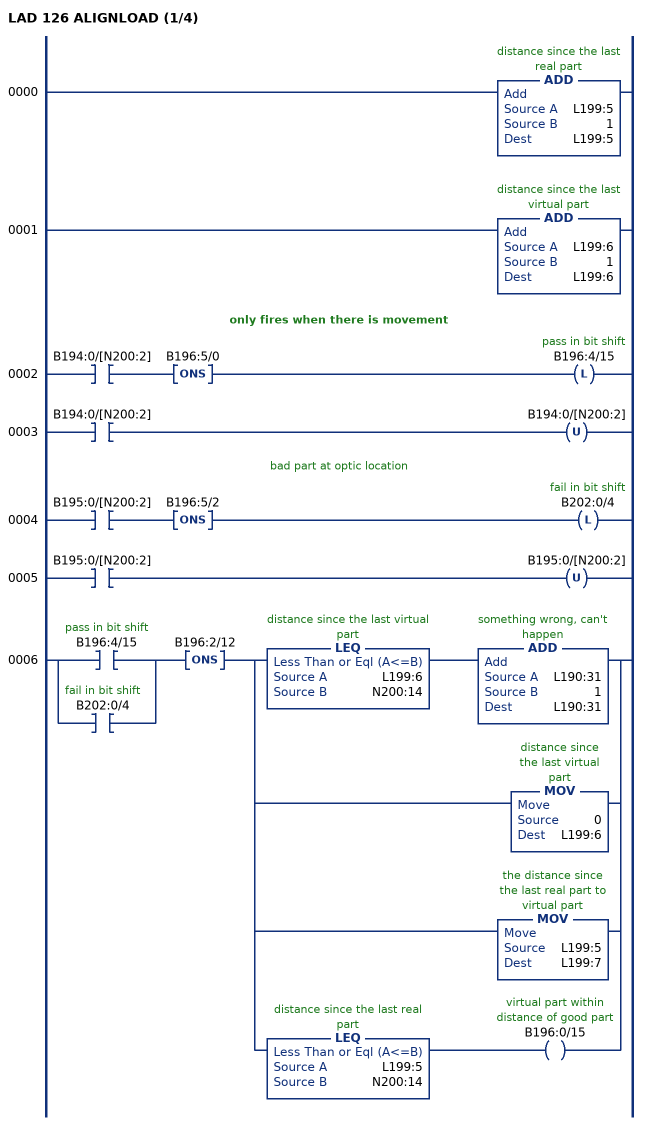
% Rung: 0 %
SOR ADD L199:5 1 L199:5 EOR
%   L199:5  "distance since the last real part" %
% Rung: 1 %
SOR ADD L199:6 1 L199:6 EOR
%   L199:6  "distance since the last virtual part" %
% Rung: 2 %
% TITLE: only fires when there is movement %
SOR XIC B194:0/[N200:2] ONS B196:5/0 OTL B196:4/15 EOR
%   N200:2  OPTIC_LOC  "top optic location" %
%   B196:4/15  "pass in bit shift" %
% Rung: 3 %
SOR XIC B194:0/[N200:2] OTU B194:0/[N200:2] EOR
%   N200:2  OPTIC_LOC  "top optic location" %
% Rung: 4 %
% bad part at optic location %
SOR XIC B195:0/[N200:2] ONS B196:5/2 OTL B202:0/4 EOR
%   N200:2  OPTIC_LOC  "top optic location" %
%   B202:0/4  "fail in bit shift" %
% Rung: 5 %
SOR XIC B195:0/[N200:2] OTU B195:0/[N200:2] EOR
%   N200:2  OPTIC_LOC  "top optic location" %
% Rung: 6 %
SOR BST XIC B196:4/15 NXB XIC B202:0/4 BND ONS B196:2/12 BST LEQ L199:6 N200:14 ADD L190:31 1 L190:31 NXB MOV 0 L199:6 NXB MOV L199:5 L199:7 NXB LEQ L199:5 N200:14 OTE B196:0/15 BND EOR
%   B196:4/15  "pass in bit shift" %
%   B202:0/4  "fail in bit shift" %
%   L199:6  "distance since the last virtual part" %
%   N200:14  "1/2 transistion zone" %
%   L190:31  "something wrong, can't happen" %
%   L199:5  "distance since the last real part" %
%   L199:7  "the distance since the last real part to virtual part" %
%   B196:0/15  "virtual part within distance of good part" %

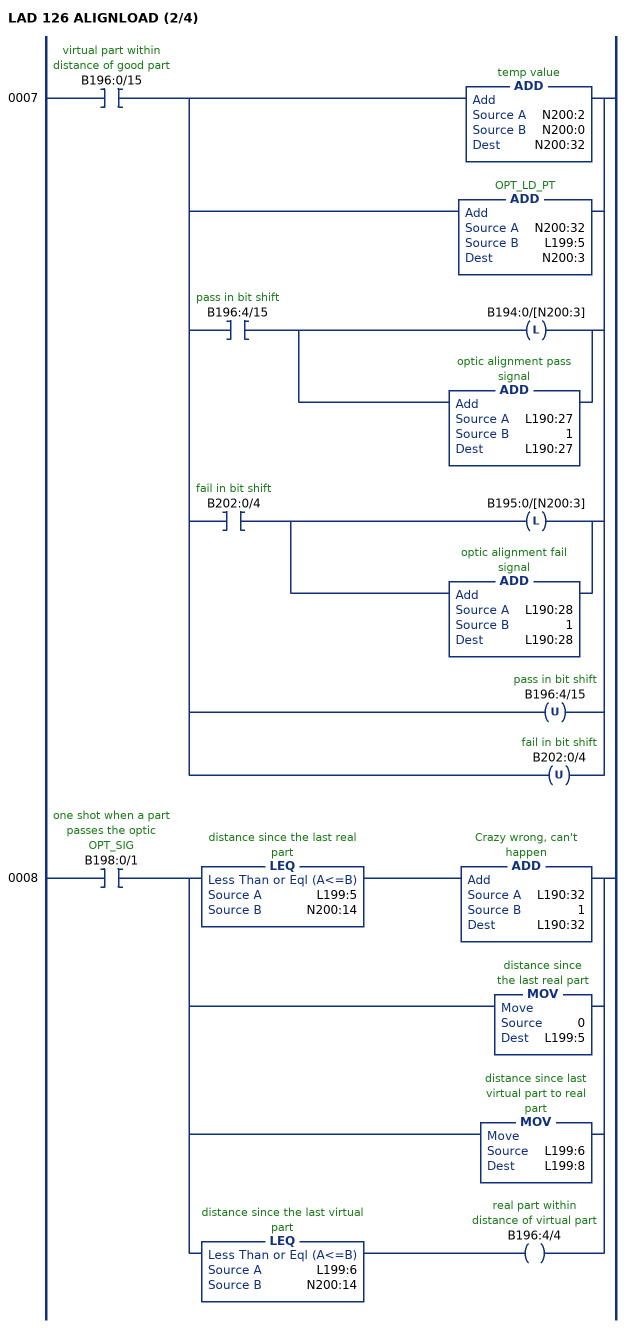
% Rung: 7 %
SOR XIC B196:0/15 BST ADD N200:2 N200:0 N200:32 NXB ADD N200:32 L199:5 N200:3 NXB XIC B196:4/15 BST OTL B194:0/[N200:3] NXB ADD L190:27 1 L190:27 BND NXB XIC B202:0/4 BST OTL B195:0/[N200:3] NXB ADD L190:28 1 L190:28 BND NXB OTU B196:4/15 NXB OTU B202:0/4 BND EOR
%   B196:0/15  "virtual part within distance of good part" %
%   N200:2  OPTIC_LOC  "top optic location" %
%   N200:0  PART_OFFSET  "1/2 part width" %
%   N200:32  "temp value" %
%   L199:5  "distance since the last real part" %
%   N200:3  OPT_LD_PT %
%   B196:4/15  "pass in bit shift" %
%   L190:27  "optic alignment pass signal" %
%   B202:0/4  "fail in bit shift" %
%   L190:28  "optic alignment fail signal" %
% Rung: 8 %
SOR XIC B198:0/1 BST LEQ L199:5 N200:14 ADD L190:32 1 L190:32 NXB MOV 0 L199:5 NXB MOV L199:6 L199:8 NXB LEQ L199:6 N200:14 OTE B196:4/4 BND EOR
%   B198:0/1  OPT_SIG  "one shot when a part passes the optic" %
%   L199:5  "distance since the last real part" %
%   N200:14  "1/2 transistion zone" %
%   L190:32  "Crazy wrong, can't happen" %
%   L199:6  "distance since the last virtual part" %
%   L199:8  "distance since last virtual part to real part" %
%   B196:4/4  "real part within distance of virtual part" %

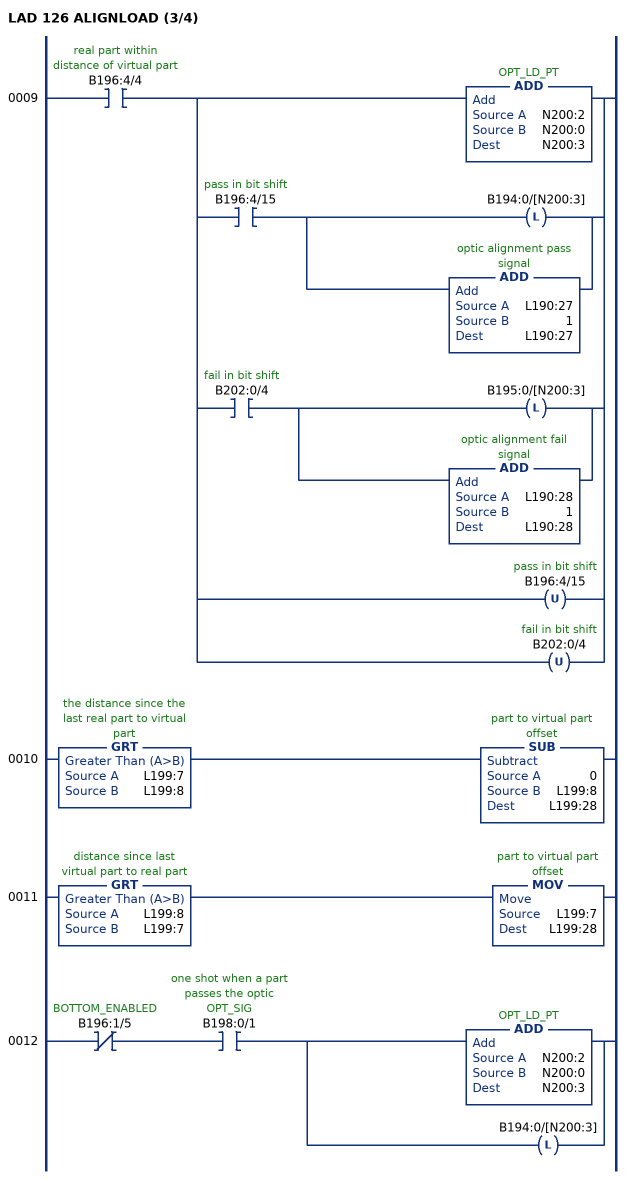
% Rung: 9 %
SOR XIC B196:4/4 BST ADD N200:2 N200:0 N200:3 NXB XIC B196:4/15 BST OTL B194:0/[N200:3] NXB ADD L190:27 1 L190:27 BND NXB XIC B202:0/4 BST OTL B195:0/[N200:3] NXB ADD L190:28 1 L190:28 BND NXB OTU B196:4/15 NXB OTU B202:0/4 BND EOR
%   B196:4/4  "real part within distance of virtual part" %
%   N200:2  OPTIC_LOC  "top optic location" %
%   N200:0  PART_OFFSET  "1/2 part width" %
%   N200:3  OPT_LD_PT %
%   B196:4/15  "pass in bit shift" %
%   L190:27  "optic alignment pass signal" %
%   B202:0/4  "fail in bit shift" %
%   L190:28  "optic alignment fail signal" %
% Rung: 10 %
SOR GRT L199:7 L199:8 SUB 0 L199:8 L199:28 EOR
%   L199:7  "the distance since the last real part to virtual part" %
%   L199:8  "distance since last virtual part to real part" %
%   L199:28  "part to virtual part offset" %
% Rung: 11 %
SOR GRT L199:8 L199:7 MOV L199:7 L199:28 EOR
%   L199:8  "distance since last virtual part to real part" %
%   L199:7  "the distance since the last real part to virtual part" %
%   L199:28  "part to virtual part offset" %
% Rung: 12 %
SOR XIO B196:1/5 XIC B198:0/1 BST ADD N200:2 N200:0 N200:3 NXB OTL B194:0/[N200:3] BND EOR
%   B196:1/5  BOTTOM_ENABLED %
%   B198:0/1  OPT_SIG  "one shot when a part passes the optic" %
%   N200:2  OPTIC_LOC  "top optic location" %
%   N200:0  PART_OFFSET  "1/2 part width" %
%   N200:3  OPT_LD_PT %

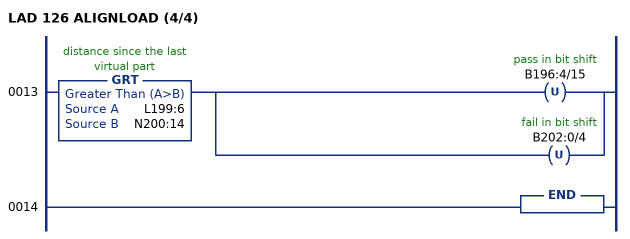
% Rung: 13 %
SOR GRT L199:6 N200:14 BST OTU B196:4/15 NXB OTU B202:0/4 BND EOR
%   L199:6  "distance since the last virtual part" %
%   N200:14  "1/2 transistion zone" %
%   B196:4/15  "pass in bit shift" %
%   B202:0/4  "fail in bit shift" %
% Rung: 14 %
SOR END EOR

LADDER 127 "NOTUSED"
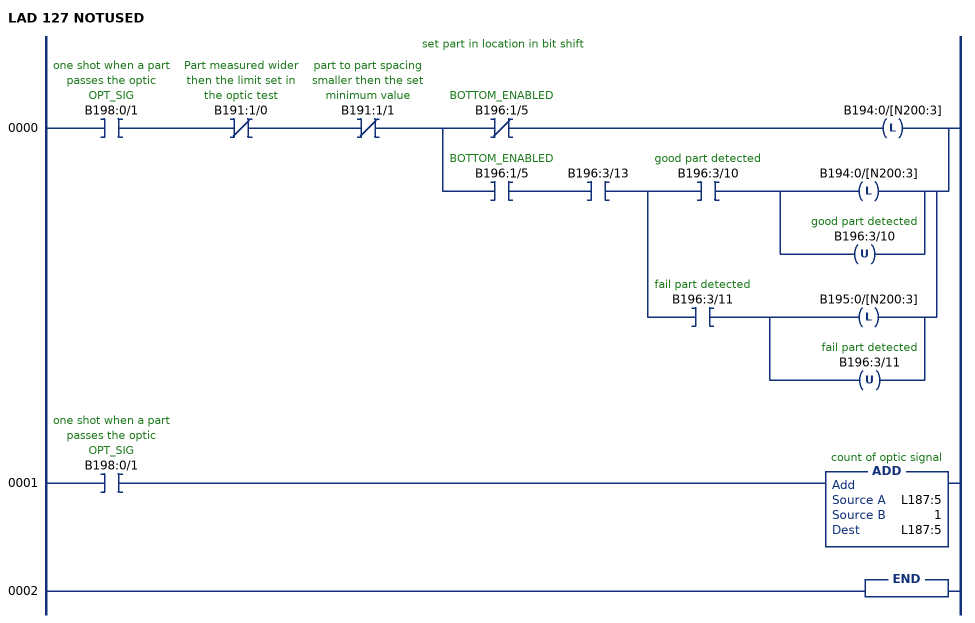
% Rung: 0 %
% set part in location in bit shift %
SOR XIC B198:0/1 XIO B191:1/0 XIO B191:1/1 BST XIO B196:1/5 OTL B194:0/[N200:3] NXB XIC B196:1/5 XIC B196:3/13 BST XIC B196:3/10 BST OTL B194:0/[N200:3] NXB OTU B196:3/10 BND NXB XIC B196:3/11 BST OTL B195:0/[N200:3] NXB OTU B196:3/11 BND BND BND EOR
%   B198:0/1  OPT_SIG  "one shot when a part passes the optic" %
%   B191:1/0  "Part measured wider then the limit set in the optic test" %
%   B191:1/1  "part to part spacing smaller then the set minimum value" %
%   B196:1/5  BOTTOM_ENABLED %
%   N200:3  OPT_LD_PT %
%   B196:3/10  "good part detected" %
%   B196:3/11  "fail part detected" %
% Rung: 1 %
SOR XIC B198:0/1 ADD L187:5 1 L187:5 EOR
%   B198:0/1  OPT_SIG  "one shot when a part passes the optic" %
%   L187:5  "count of optic signal" %
% Rung: 2 %
SOR END EOR

LADDER 128 "NOTUSED3"
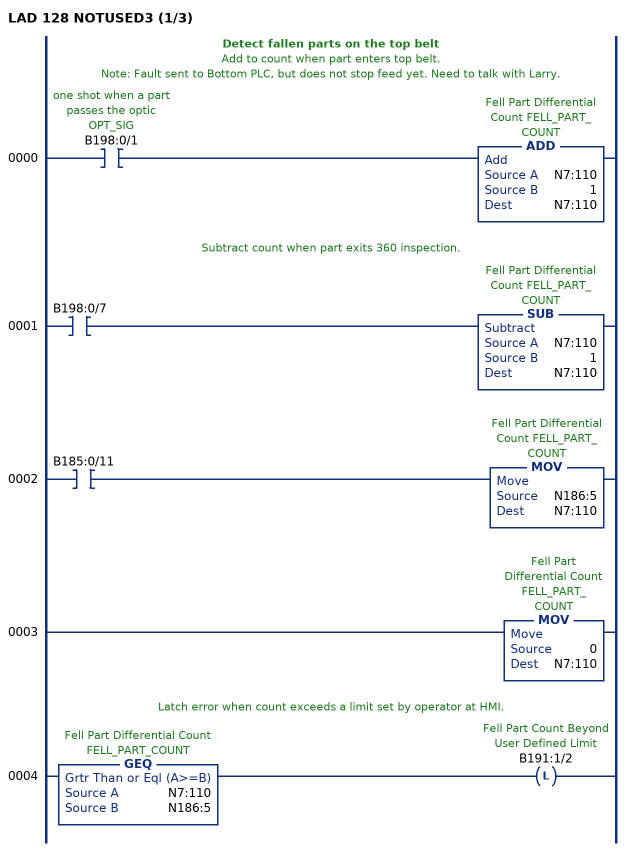
% Rung: 0 %
% TITLE: Detect fallen parts on the top belt %
% Add to count when part enters top belt.
% Note: Fault sent to Bottom PLC, but does not stop feed yet. Need to talk with Larry. %
SOR XIC B198:0/1 ADD N7:110 1 N7:110 EOR
%   B198:0/1  OPT_SIG  "one shot when a part passes the optic" %
%   N7:110  FELL_PART_COUNT  "Fell Part Differential Count" %
% Rung: 1 %
% Subtract count when part exits 360 inspection. %
SOR XIC B198:0/7 SUB N7:110 1 N7:110 EOR
%   N7:110  FELL_PART_COUNT  "Fell Part Differential Count" %
% Rung: 2 %
SOR XIC B185:0/11 MOV N186:5 N7:110 EOR
%   N186:5  FELL_PART_LIMIT  "Fell Part Differential Limit From HMI" %
%   N7:110  FELL_PART_COUNT  "Fell Part Differential Count" %
% Rung: 3 %
SOR MOV 0 N7:110 EOR
%   N7:110  FELL_PART_COUNT  "Fell Part Differential Count" %
% Rung: 4 %
% Latch error when count exceeds a limit set by operator at HMI. %
SOR GEQ N7:110 N186:5 OTL B191:1/2 EOR
%   N7:110  FELL_PART_COUNT  "Fell Part Differential Count" %
%   N186:5  FELL_PART_LIMIT  "Fell Part Differential Limit From HMI" %
%   B191:1/2  "Fell Part Count Beyond User Defined Limit" %

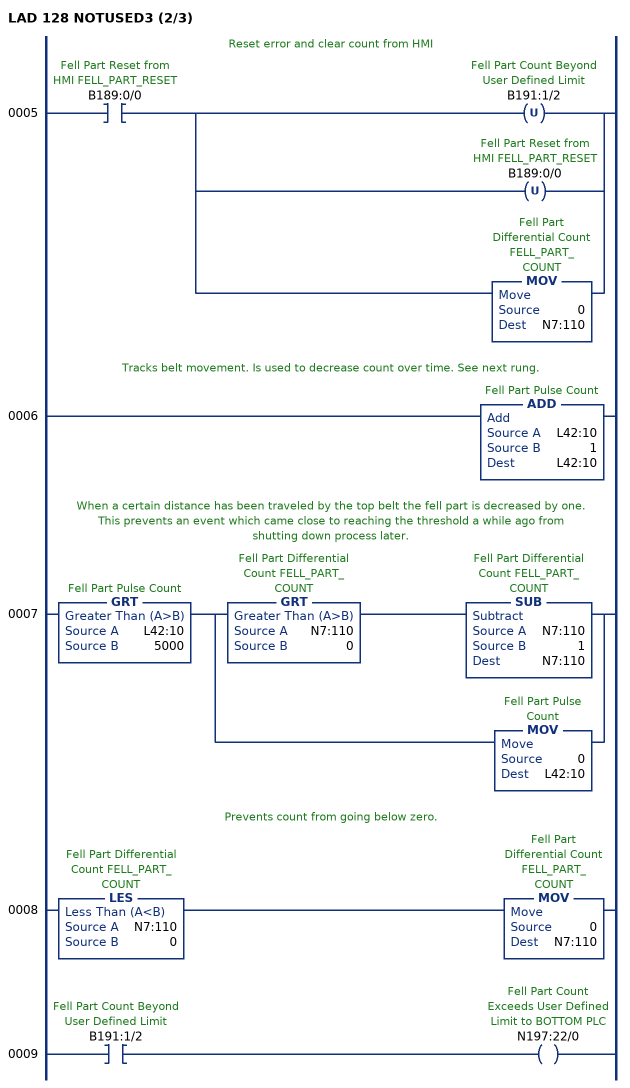
% Rung: 5 %
% Reset error and clear count from HMI %
SOR XIC B189:0/0 BST OTU B191:1/2 NXB OTU B189:0/0 NXB MOV 0 N7:110 BND EOR
%   B189:0/0  FELL_PART_RESET  "Fell Part Reset from HMI" %
%   B191:1/2  "Fell Part Count Beyond User Defined Limit" %
%   N7:110  FELL_PART_COUNT  "Fell Part Differential Count" %
% Rung: 6 %
% Tracks belt movement. Is used to decrease count over time. See next rung. %
SOR ADD L42:10 1 L42:10 EOR
%   L42:10  "Fell Part Pulse Count" %
% Rung: 7 %
% When a certain distance has been traveled by the top belt the fell part is decreased by one. This prevents an event which came close to reaching the threshold a while ago from shutting down process later. %
SOR GRT L42:10 5000 BST GRT N7:110 0 SUB N7:110 1 N7:110 NXB MOV 0 L42:10 BND EOR
%   L42:10  "Fell Part Pulse Count" %
%   N7:110  FELL_PART_COUNT  "Fell Part Differential Count" %
% Rung: 8 %
% Prevents count from going below zero. %
SOR LES N7:110 0 MOV 0 N7:110 EOR
%   N7:110  FELL_PART_COUNT  "Fell Part Differential Count" %
% Rung: 9 %
SOR XIC B191:1/2 OTE N197:22/0 EOR
%   B191:1/2  "Fell Part Count Beyond User Defined Limit" %
%   N197:22/0  "Fell Part Count Exceeds User Defined Limit to BOTTOM PLC" %

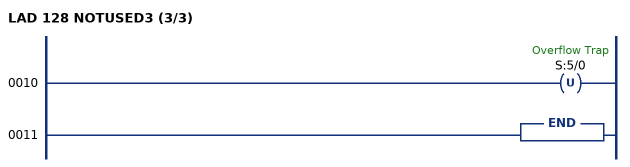
% Rung: 10 %
SOR OTU S:5/0 EOR
%   S:5/0  "Overflow Trap" %
% Rung: 11 %
SOR END EOR

LADDER 130 "INS 5 TRIG"
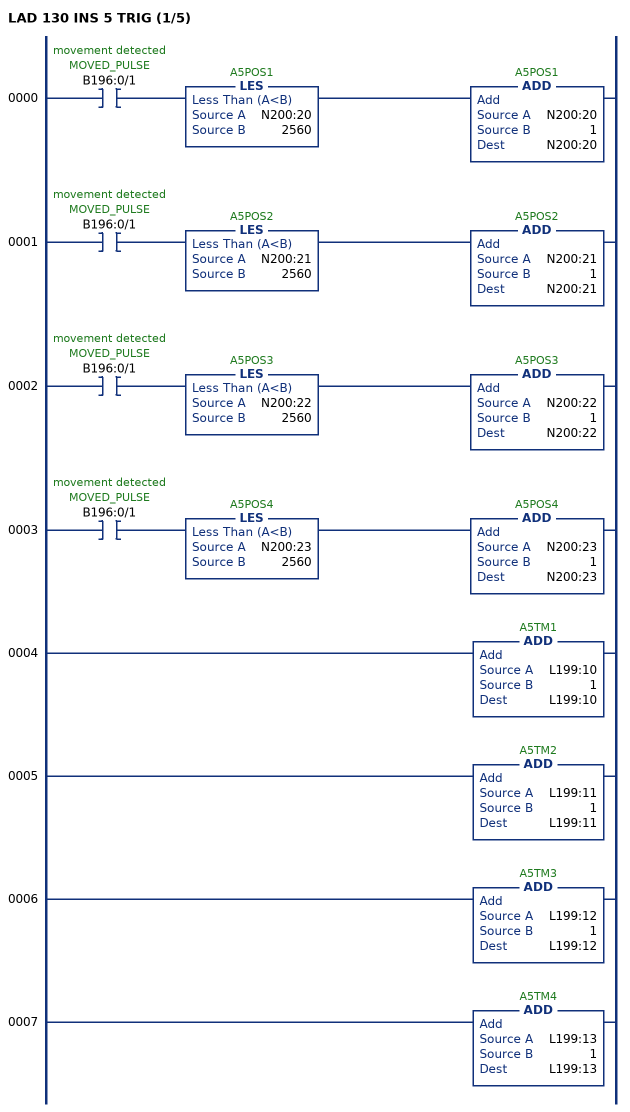
% Rung: 0 %
SOR XIC B196:0/1 LES N200:20 2560 ADD N200:20 1 N200:20 EOR
%   B196:0/1  MOVED_PULSE  "movement detected" %
%   N200:20  A5POS1 %
% Rung: 1 %
SOR XIC B196:0/1 LES N200:21 2560 ADD N200:21 1 N200:21 EOR
%   B196:0/1  MOVED_PULSE  "movement detected" %
%   N200:21  A5POS2 %
% Rung: 2 %
SOR XIC B196:0/1 LES N200:22 2560 ADD N200:22 1 N200:22 EOR
%   B196:0/1  MOVED_PULSE  "movement detected" %
%   N200:22  A5POS3 %
% Rung: 3 %
SOR XIC B196:0/1 LES N200:23 2560 ADD N200:23 1 N200:23 EOR
%   B196:0/1  MOVED_PULSE  "movement detected" %
%   N200:23  A5POS4 %
% Rung: 4 %
SOR ADD L199:10 1 L199:10 EOR
%   L199:10  A5TM1 %
% Rung: 5 %
SOR ADD L199:11 1 L199:11 EOR
%   L199:11  A5TM2 %
% Rung: 6 %
SOR ADD L199:12 1 L199:12 EOR
%   L199:12  A5TM3 %
% Rung: 7 %
SOR ADD L199:13 1 L199:13 EOR
%   L199:13  A5TM4 %

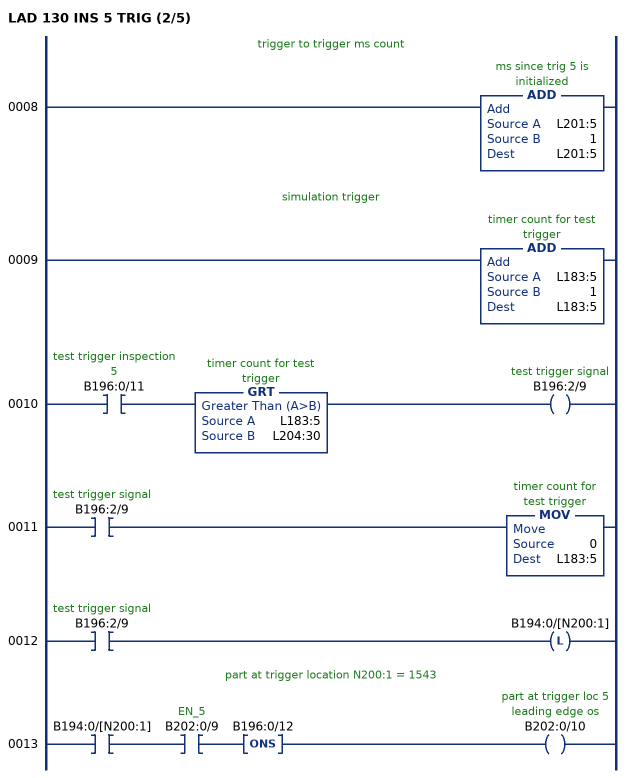
% Rung: 8 %
% trigger to trigger ms count %
SOR ADD L201:5 1 L201:5 EOR
%   L201:5  "ms since trig 5 is initialized" %
% Rung: 9 %
% simulation trigger %
SOR ADD L183:5 1 L183:5 EOR
%   L183:5  "timer count for test trigger" %
% Rung: 10 %
SOR XIC B196:0/11 GRT L183:5 L204:30 OTE B196:2/9 EOR
%   B196:0/11  "test trigger inspection 5" %
%   L183:5  "timer count for test trigger" %
%   B196:2/9  "test trigger signal" %
% Rung: 11 %
SOR XIC B196:2/9 MOV 0 L183:5 EOR
%   B196:2/9  "test trigger signal" %
%   L183:5  "timer count for test trigger" %
% Rung: 12 %
SOR XIC B196:2/9 OTL B194:0/[N200:1] EOR
%   B196:2/9  "test trigger signal" %
%   N200:1  INS_5_TRIG_LOC %
% Rung: 13 %
% part at trigger location N200:1 = 1543 %
SOR XIC B194:0/[N200:1] XIC B202:0/9 ONS B196:0/12 OTE B202:0/10 EOR
%   N200:1  INS_5_TRIG_LOC %
%   B202:0/9  EN_5 %
%   B202:0/10  "part at trigger loc 5 leading edge os" %

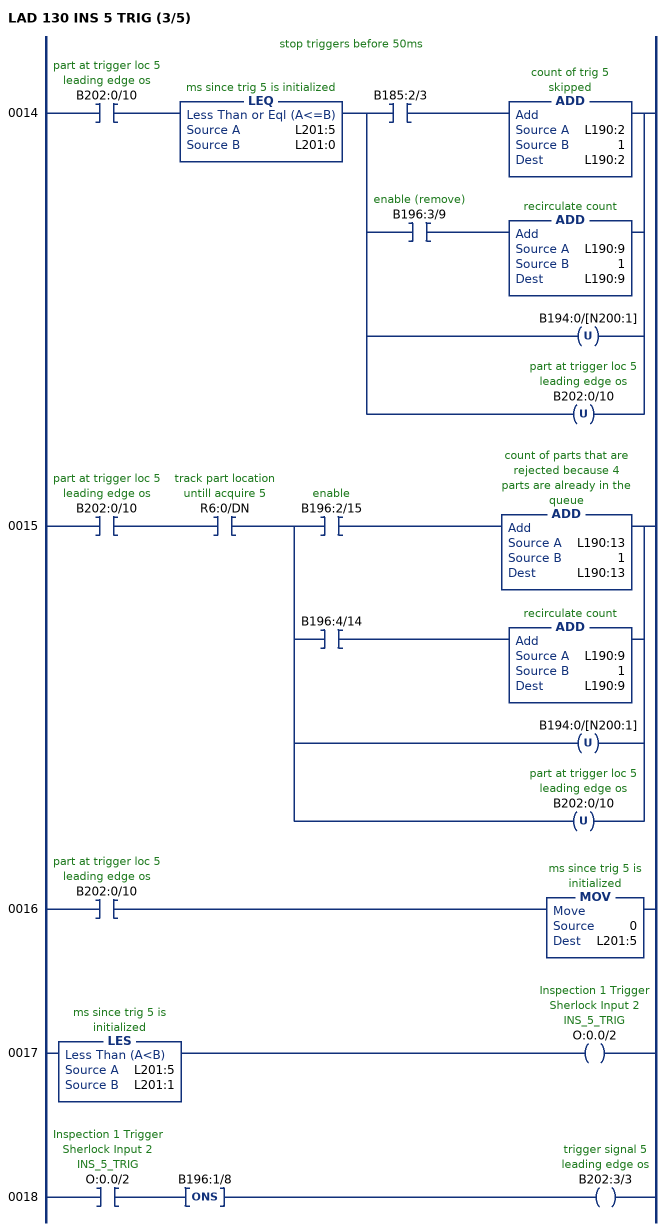
% Rung: 14 %
% stop triggers before 50ms %
SOR XIC B202:0/10 LEQ L201:5 L201:0 BST XIC B185:2/3 ADD L190:2 1 L190:2 NXB XIC B196:3/9 ADD L190:9 1 L190:9 NXB OTU B194:0/[N200:1] NXB OTU B202:0/10 BND EOR
%   B202:0/10  "part at trigger loc 5 leading edge os" %
%   L201:5  "ms since trig 5 is initialized" %
%   L201:0  CAM_5_MIN_CYCLE_TIME %
%   L190:2  "count of trig 5 skipped" %
%   B196:3/9  "enable (remove)" %
%   L190:9  "recirculate count" %
%   N200:1  INS_5_TRIG_LOC %
% Rung: 15 %
SOR XIC B202:0/10 XIC R6:0/DN BST XIC B196:2/15 ADD L190:13 1 L190:13 NXB XIC B196:4/14 ADD L190:9 1 L190:9 NXB OTU B194:0/[N200:1] NXB OTU B202:0/10 BND EOR
%   B202:0/10  "part at trigger loc 5 leading edge os" %
%   R6:0  "track part location untill acquire 5" %
%   B196:2/15  "enable" %
%   L190:13  "count of parts that are rejected because 4 parts are already in the queue" %
%   L190:9  "recirculate count" %
%   N200:1  INS_5_TRIG_LOC %
% Rung: 16 %
SOR XIC B202:0/10 MOV 0 L201:5 EOR
%   B202:0/10  "part at trigger loc 5 leading edge os" %
%   L201:5  "ms since trig 5 is initialized" %
% Rung: 17 %
SOR LES L201:5 L201:1 OTE O:0.0/2 EOR
%   L201:5  "ms since trig 5 is initialized" %
%   L201:1  CAM_5_TRIG_TIME %
%   O:0.0/2  INS_5_TRIG  "Inspection 1 Trigger Sherlock Input 2" %
% Rung: 18 %
SOR XIC O:0.0/2 ONS B196:1/8 OTE B202:3/3 EOR
%   O:0.0/2  INS_5_TRIG  "Inspection 1 Trigger Sherlock Input 2" %
%   B202:3/3  "trigger signal 5 leading edge os" %

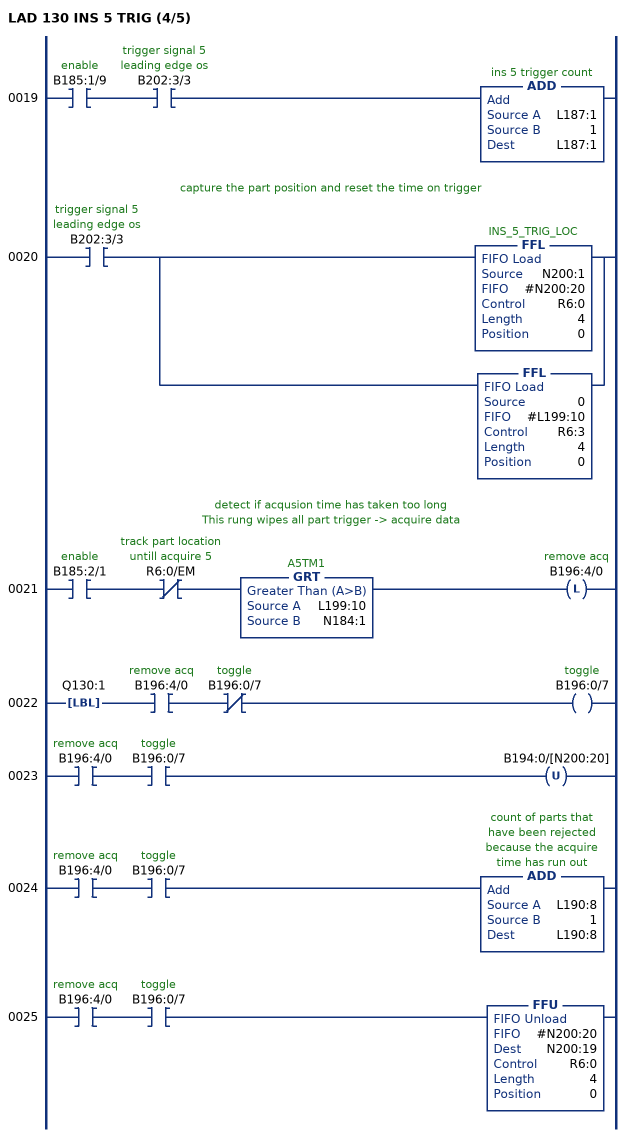
% Rung: 19 %
SOR XIC B185:1/9 XIC B202:3/3 ADD L187:1 1 L187:1 EOR
%   B185:1/9  "enable" %
%   B202:3/3  "trigger signal 5 leading edge os" %
%   L187:1  "ins 5 trigger count" %
% Rung: 20 %
% capture the part position and reset the time on trigger %
SOR XIC B202:3/3 BST FFL N200:1 #N200:20 R6:0 4 0 NXB FFL 0 #L199:10 R6:3 4 0 BND EOR
%   B202:3/3  "trigger signal 5 leading edge os" %
%   N200:1  INS_5_TRIG_LOC %
%   N200:20  A5POS1 %
%   R6:0  "track part location untill acquire 5" %
%   L199:10  A5TM1 %
%   R6:3  "track acquire time 5" %
% Rung: 21 %
% detect if acqusion time has taken too long
% This rung wipes all part trigger -> acquire data %
SOR XIC B185:2/1 XIO R6:0/EM GRT L199:10 N184:1 OTL B196:4/0 EOR
%   B185:2/1  "enable" %
%   R6:0  "track part location untill acquire 5" %
%   L199:10  A5TM1 %
%   N184:1  "maximum acquire time 5" %
%   B196:4/0  "remove acq" %
% Rung: 22 %
SOR LBL Q130:1 XIC B196:4/0 XIO B196:0/7 OTE B196:0/7 EOR
%   B196:4/0  "remove acq" %
%   B196:0/7  "toggle" %
% Rung: 23 %
SOR XIC B196:4/0 XIC B196:0/7 OTU B194:0/[N200:20] EOR
%   B196:4/0  "remove acq" %
%   B196:0/7  "toggle" %
%   N200:20  A5POS1 %
% Rung: 24 %
SOR XIC B196:4/0 XIC B196:0/7 ADD L190:8 1 L190:8 EOR
%   B196:4/0  "remove acq" %
%   B196:0/7  "toggle" %
%   L190:8  "count of parts that have been rejected because the acquire time has run out" %
% Rung: 25 %
SOR XIC B196:4/0 XIC B196:0/7 FFU #N200:20 N200:19 R6:0 4 0 EOR
%   B196:4/0  "remove acq" %
%   B196:0/7  "toggle" %
%   N200:20  A5POS1 %
%   R6:0  "track part location untill acquire 5" %

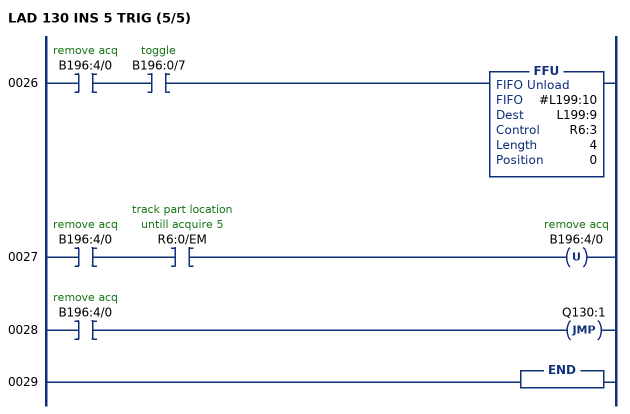
% Rung: 26 %
SOR XIC B196:4/0 XIC B196:0/7 FFU #L199:10 L199:9 R6:3 4 0 EOR
%   B196:4/0  "remove acq" %
%   B196:0/7  "toggle" %
%   L199:10  A5TM1 %
%   R6:3  "track acquire time 5" %
% Rung: 27 %
SOR XIC B196:4/0 XIC R6:0/EM OTU B196:4/0 EOR
%   B196:4/0  "remove acq" %
%   R6:0  "track part location untill acquire 5" %
% Rung: 28 %
SOR XIC B196:4/0 JMP Q130:1 EOR
%   B196:4/0  "remove acq" %
% Rung: 29 %
SOR END EOR

LADDER 131 "INS 5 RSLT"
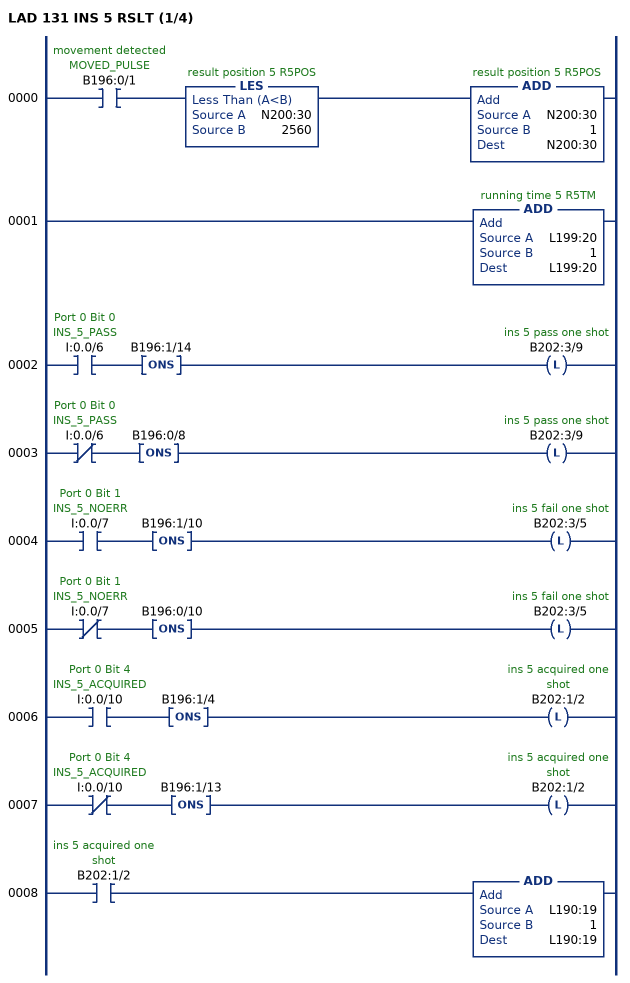
% Rung: 0 %
SOR XIC B196:0/1 LES N200:30 2560 ADD N200:30 1 N200:30 EOR
%   B196:0/1  MOVED_PULSE  "movement detected" %
%   N200:30  R5POS  "result position 5" %
% Rung: 1 %
SOR ADD L199:20 1 L199:20 EOR
%   L199:20  R5TM  "running time 5" %
% Rung: 2 %
SOR XIC I:0.0/6 ONS B196:1/14 OTL B202:3/9 EOR
%   I:0.0/6  INS_5_PASS  "Port 0 Bit 0" %
%   B202:3/9  "ins 5 pass one shot" %
% Rung: 3 %
SOR XIO I:0.0/6 ONS B196:0/8 OTL B202:3/9 EOR
%   I:0.0/6  INS_5_PASS  "Port 0 Bit 0" %
%   B202:3/9  "ins 5 pass one shot" %
% Rung: 4 %
SOR XIC I:0.0/7 ONS B196:1/10 OTL B202:3/5 EOR
%   I:0.0/7  INS_5_NOERR  "Port 0 Bit 1" %
%   B202:3/5  "ins 5 fail one shot" %
% Rung: 5 %
SOR XIO I:0.0/7 ONS B196:0/10 OTL B202:3/5 EOR
%   I:0.0/7  INS_5_NOERR  "Port 0 Bit 1" %
%   B202:3/5  "ins 5 fail one shot" %
% Rung: 6 %
SOR XIC I:0.0/10 ONS B196:1/4 OTL B202:1/2 EOR
%   I:0.0/10  INS_5_ACQUIRED  "Port 0 Bit 4" %
%   B202:1/2  "ins 5 acquired one shot" %
% Rung: 7 %
SOR XIO I:0.0/10 ONS B196:1/13 OTL B202:1/2 EOR
%   I:0.0/10  INS_5_ACQUIRED  "Port 0 Bit 4" %
%   B202:1/2  "ins 5 acquired one shot" %
% Rung: 8 %
SOR XIC B202:1/2 ADD L190:19 1 L190:19 EOR
%   B202:1/2  "ins 5 acquired one shot" %

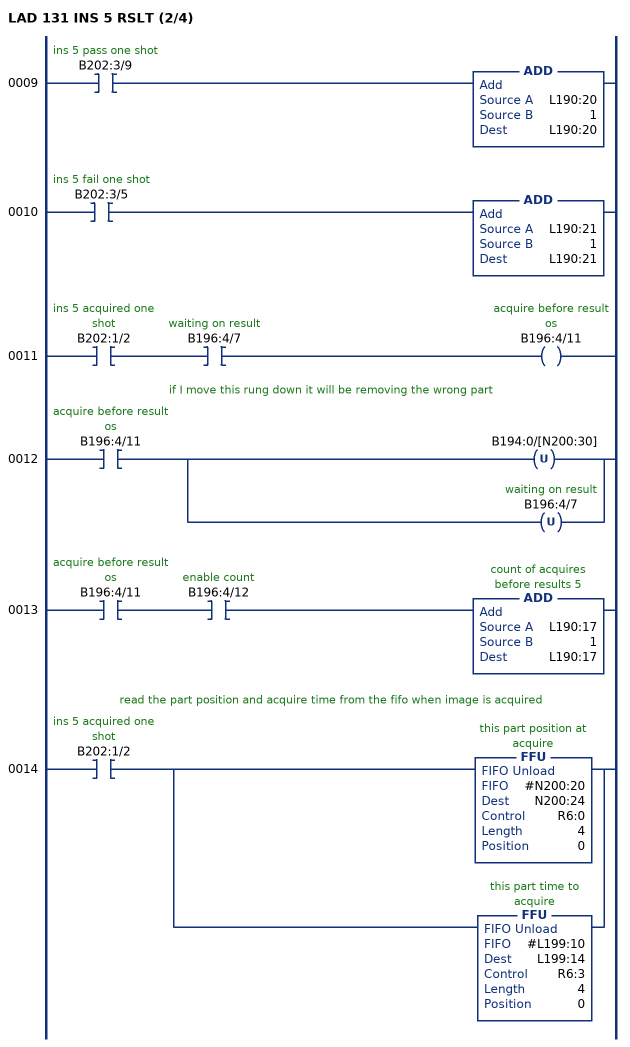
% Rung: 9 %
SOR XIC B202:3/9 ADD L190:20 1 L190:20 EOR
%   B202:3/9  "ins 5 pass one shot" %
% Rung: 10 %
SOR XIC B202:3/5 ADD L190:21 1 L190:21 EOR
%   B202:3/5  "ins 5 fail one shot" %
% Rung: 11 %
SOR XIC B202:1/2 XIC B196:4/7 OTE B196:4/11 EOR
%   B202:1/2  "ins 5 acquired one shot" %
%   B196:4/7  "waiting on result" %
%   B196:4/11  "acquire before result os" %
% Rung: 12 %
% if I move this rung down it will be removing the wrong part %
SOR XIC B196:4/11 BST OTU B194:0/[N200:30] NXB OTU B196:4/7 BND EOR
%   B196:4/11  "acquire before result os" %
%   N200:30  R5POS  "result position 5" %
%   B196:4/7  "waiting on result" %
% Rung: 13 %
SOR XIC B196:4/11 XIC B196:4/12 ADD L190:17 1 L190:17 EOR
%   B196:4/11  "acquire before result os" %
%   B196:4/12  "enable count" %
%   L190:17  "count of acquires before results 5" %
% Rung: 14 %
% read the part position and acquire time from the fifo when image is acquired %
SOR XIC B202:1/2 BST FFU #N200:20 N200:24 R6:0 4 0 NXB FFU #L199:10 L199:14 R6:3 4 0 BND EOR
%   B202:1/2  "ins 5 acquired one shot" %
%   N200:20  A5POS1 %
%   N200:24  "this part position at acquire" %
%   R6:0  "track part location untill acquire 5" %
%   L199:10  A5TM1 %
%   L199:14  "this part time to acquire" %
%   R6:3  "track acquire time 5" %

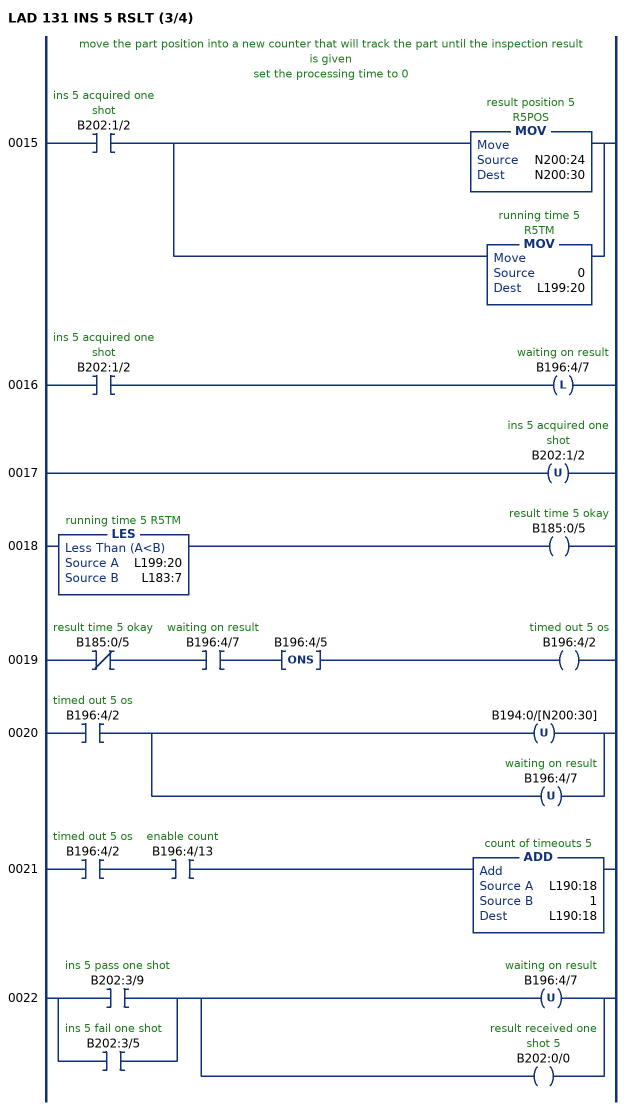
% Rung: 15 %
% move the part position into a new counter that will track the part until the inspection result is given
% set the processing time to 0 %
SOR XIC B202:1/2 BST MOV N200:24 N200:30 NXB MOV 0 L199:20 BND EOR
%   B202:1/2  "ins 5 acquired one shot" %
%   N200:24  "this part position at acquire" %
%   N200:30  R5POS  "result position 5" %
%   L199:20  R5TM  "running time 5" %
% Rung: 16 %
SOR XIC B202:1/2 OTL B196:4/7 EOR
%   B202:1/2  "ins 5 acquired one shot" %
%   B196:4/7  "waiting on result" %
% Rung: 17 %
SOR OTU B202:1/2 EOR
%   B202:1/2  "ins 5 acquired one shot" %
% Rung: 18 %
SOR LES L199:20 L183:7 OTE B185:0/5 EOR
%   L199:20  R5TM  "running time 5" %
%   L183:7  "max process time 5" %
%   B185:0/5  "result time 5 okay" %
% Rung: 19 %
SOR XIO B185:0/5 XIC B196:4/7 ONS B196:4/5 OTE B196:4/2 EOR
%   B185:0/5  "result time 5 okay" %
%   B196:4/7  "waiting on result" %
%   B196:4/2  "timed out 5 os" %
% Rung: 20 %
SOR XIC B196:4/2 BST OTU B194:0/[N200:30] NXB OTU B196:4/7 BND EOR
%   B196:4/2  "timed out 5 os" %
%   N200:30  R5POS  "result position 5" %
%   B196:4/7  "waiting on result" %
% Rung: 21 %
SOR XIC B196:4/2 XIC B196:4/13 ADD L190:18 1 L190:18 EOR
%   B196:4/2  "timed out 5 os" %
%   B196:4/13  "enable count" %
%   L190:18  "count of timeouts 5" %
% Rung: 22 %
SOR BST XIC B202:3/9 NXB XIC B202:3/5 BND BST OTU B196:4/7 NXB OTE B202:0/0 BND EOR
%   B202:3/9  "ins 5 pass one shot" %
%   B202:3/5  "ins 5 fail one shot" %
%   B196:4/7  "waiting on result" %
%   B202:0/0  "result received one shot 5" %

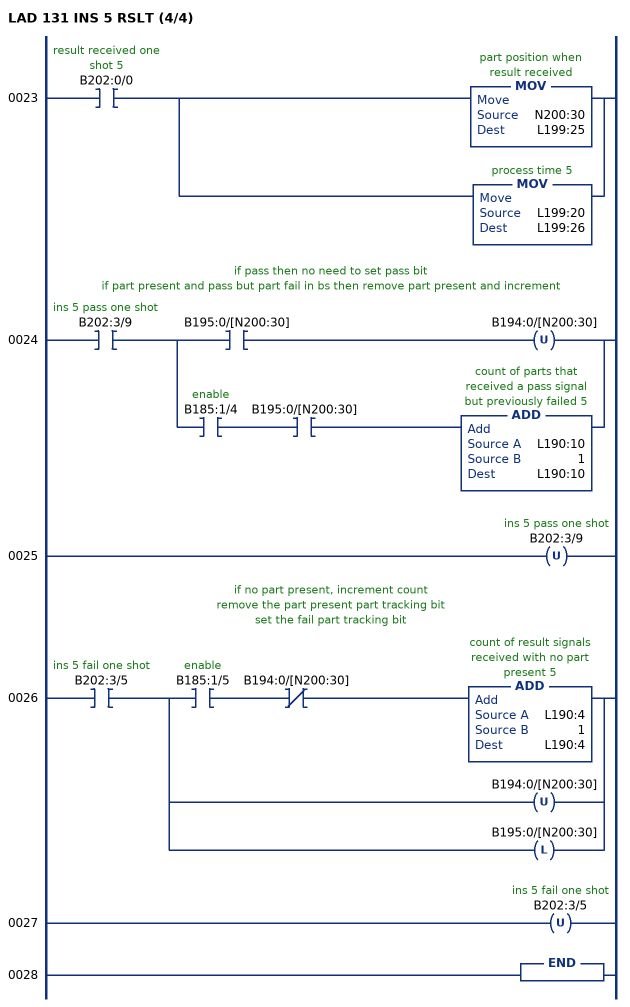
% Rung: 23 %
SOR XIC B202:0/0 BST MOV N200:30 L199:25 NXB MOV L199:20 L199:26 BND EOR
%   B202:0/0  "result received one shot 5" %
%   N200:30  R5POS  "result position 5" %
%   L199:25  "part position when result received" %
%   L199:20  R5TM  "running time 5" %
%   L199:26  "process time 5" %
% Rung: 24 %
% if pass then no need to set pass bit
% if part present and pass but part fail in bs then remove part present and increment %
SOR XIC B202:3/9 BST XIC B195:0/[N200:30] OTU B194:0/[N200:30] NXB XIC B185:1/4 XIC B195:0/[N200:30] ADD L190:10 1 L190:10 BND EOR
%   B202:3/9  "ins 5 pass one shot" %
%   N200:30  R5POS  "result position 5" %
%   B185:1/4  "enable" %
%   L190:10  "count of parts that received a pass signal but previously failed 5" %
% Rung: 25 %
SOR OTU B202:3/9 EOR
%   B202:3/9  "ins 5 pass one shot" %
% Rung: 26 %
% if no part present, increment count
% remove the part present part tracking bit
% set the fail part tracking bit %
SOR XIC B202:3/5 BST XIC B185:1/5 XIO B194:0/[N200:30] ADD L190:4 1 L190:4 NXB OTU B194:0/[N200:30] NXB OTL B195:0/[N200:30] BND EOR
%   B202:3/5  "ins 5 fail one shot" %
%   B185:1/5  "enable" %
%   N200:30  R5POS  "result position 5" %
%   L190:4  "count of result signals received with no part present 5" %
% Rung: 27 %
SOR OTU B202:3/5 EOR
%   B202:3/5  "ins 5 fail one shot" %
% Rung: 28 %
SOR END EOR

LADDER 140 "INS 6 TRIG"
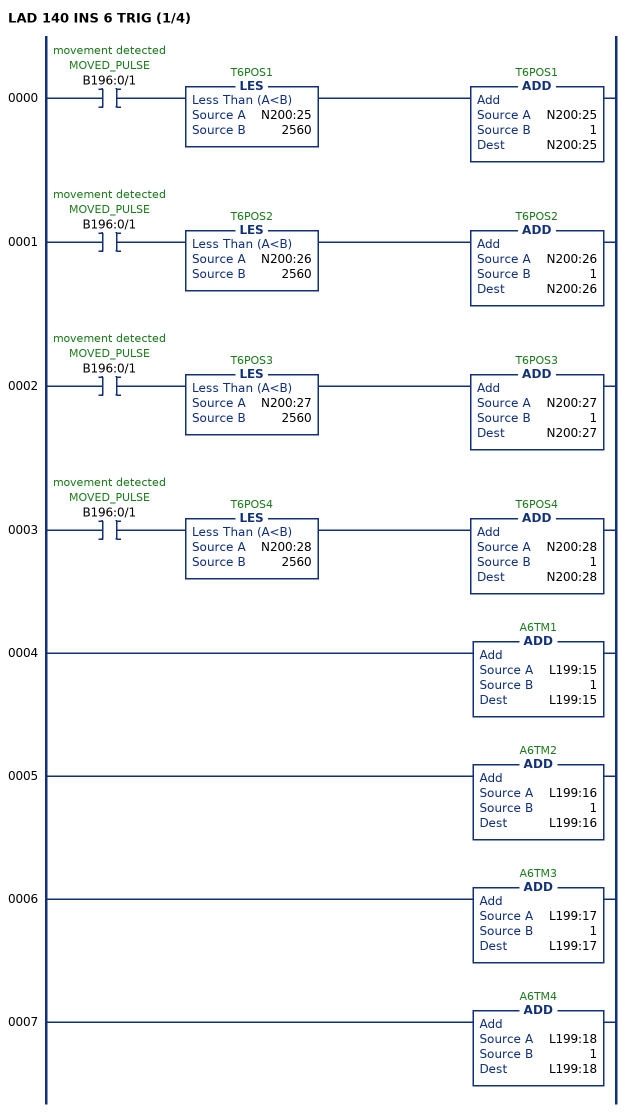
% Rung: 0 %
SOR XIC B196:0/1 LES N200:25 2560 ADD N200:25 1 N200:25 EOR
%   B196:0/1  MOVED_PULSE  "movement detected" %
%   N200:25  T6POS1 %
% Rung: 1 %
SOR XIC B196:0/1 LES N200:26 2560 ADD N200:26 1 N200:26 EOR
%   B196:0/1  MOVED_PULSE  "movement detected" %
%   N200:26  T6POS2 %
% Rung: 2 %
SOR XIC B196:0/1 LES N200:27 2560 ADD N200:27 1 N200:27 EOR
%   B196:0/1  MOVED_PULSE  "movement detected" %
%   N200:27  T6POS3 %
% Rung: 3 %
SOR XIC B196:0/1 LES N200:28 2560 ADD N200:28 1 N200:28 EOR
%   B196:0/1  MOVED_PULSE  "movement detected" %
%   N200:28  T6POS4 %
% Rung: 4 %
SOR ADD L199:15 1 L199:15 EOR
%   L199:15  A6TM1 %
% Rung: 5 %
SOR ADD L199:16 1 L199:16 EOR
%   L199:16  A6TM2 %
% Rung: 6 %
SOR ADD L199:17 1 L199:17 EOR
%   L199:17  A6TM3 %
% Rung: 7 %
SOR ADD L199:18 1 L199:18 EOR
%   L199:18  A6TM4 %

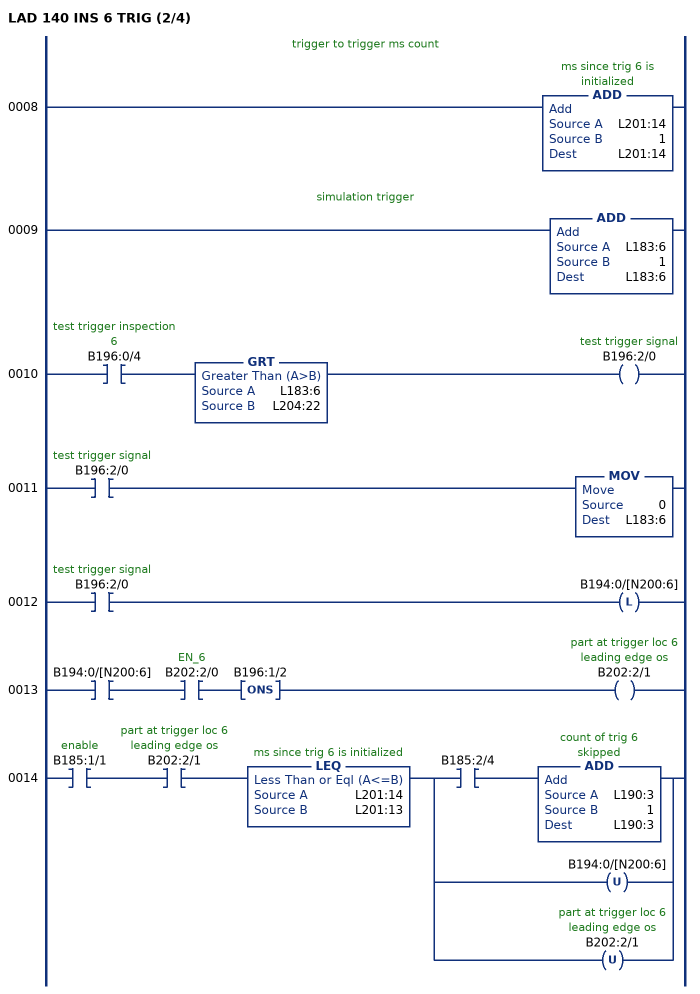
% Rung: 8 %
% trigger to trigger ms count %
SOR ADD L201:14 1 L201:14 EOR
%   L201:14  "ms since trig 6 is initialized" %
% Rung: 9 %
% simulation trigger %
SOR ADD L183:6 1 L183:6 EOR
% Rung: 10 %
SOR XIC B196:0/4 GRT L183:6 L204:22 OTE B196:2/0 EOR
%   B196:0/4  "test trigger inspection 6" %
%   B196:2/0  "test trigger signal" %
% Rung: 11 %
SOR XIC B196:2/0 MOV 0 L183:6 EOR
%   B196:2/0  "test trigger signal" %
% Rung: 12 %
SOR XIC B196:2/0 OTL B194:0/[N200:6] EOR
%   B196:2/0  "test trigger signal" %
%   N200:6  INS_6_TRIG_LOC %
% Rung: 13 %
SOR XIC B194:0/[N200:6] XIC B202:2/0 ONS B196:1/2 OTE B202:2/1 EOR
%   N200:6  INS_6_TRIG_LOC %
%   B202:2/0  EN_6 %
%   B202:2/1  "part at trigger loc 6 leading edge os" %
% Rung: 14 %
SOR XIC B185:1/1 XIC B202:2/1 LEQ L201:14 L201:13 BST XIC B185:2/4 ADD L190:3 1 L190:3 NXB OTU B194:0/[N200:6] NXB OTU B202:2/1 BND EOR
%   B185:1/1  "enable" %
%   B202:2/1  "part at trigger loc 6 leading edge os" %
%   L201:14  "ms since trig 6 is initialized" %
%   L201:13  CAM_6_MIN_CYCLE_TIME %
%   L190:3  "count of trig 6 skipped" %
%   N200:6  INS_6_TRIG_LOC %

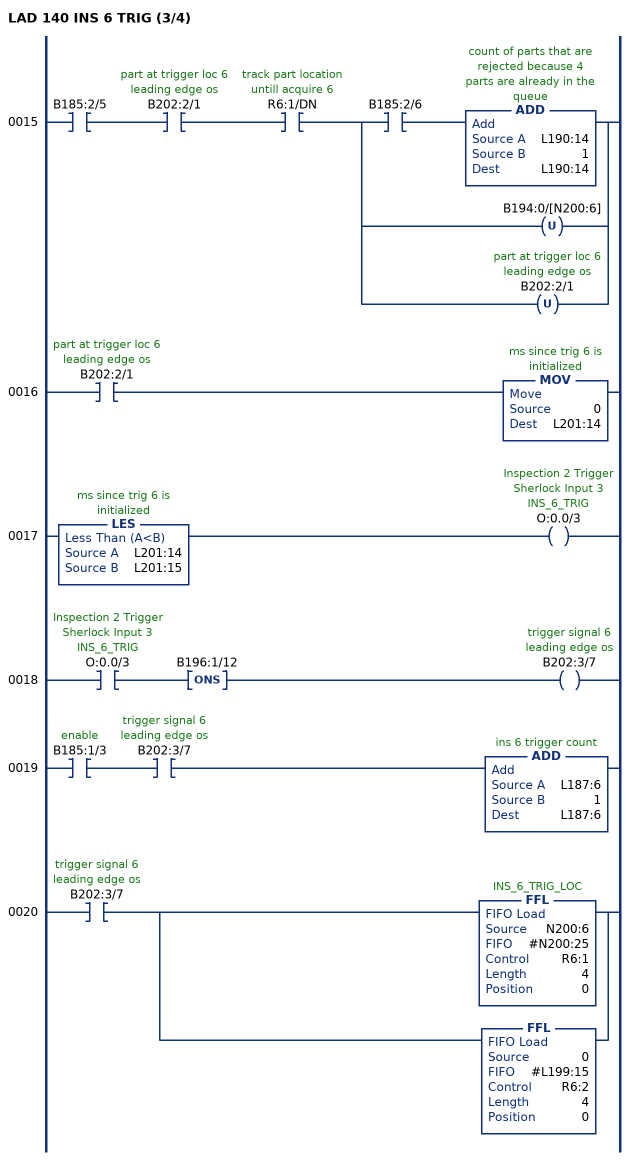
% Rung: 15 %
SOR XIC B185:2/5 XIC B202:2/1 XIC R6:1/DN BST XIC B185:2/6 ADD L190:14 1 L190:14 NXB OTU B194:0/[N200:6] NXB OTU B202:2/1 BND EOR
%   B202:2/1  "part at trigger loc 6 leading edge os" %
%   R6:1  "track part location untill acquire 6" %
%   L190:14  "count of parts that are rejected because 4 parts are already in the queue" %
%   N200:6  INS_6_TRIG_LOC %
% Rung: 16 %
SOR XIC B202:2/1 MOV 0 L201:14 EOR
%   B202:2/1  "part at trigger loc 6 leading edge os" %
%   L201:14  "ms since trig 6 is initialized" %
% Rung: 17 %
SOR LES L201:14 L201:15 OTE O:0.0/3 EOR
%   L201:14  "ms since trig 6 is initialized" %
%   L201:15  CAM_6_TRIG_TIME %
%   O:0.0/3  INS_6_TRIG  "Inspection 2 Trigger Sherlock Input 3" %
% Rung: 18 %
SOR XIC O:0.0/3 ONS B196:1/12 OTE B202:3/7 EOR
%   O:0.0/3  INS_6_TRIG  "Inspection 2 Trigger Sherlock Input 3" %
%   B202:3/7  "trigger signal 6 leading edge os" %
% Rung: 19 %
SOR XIC B185:1/3 XIC B202:3/7 ADD L187:6 1 L187:6 EOR
%   B185:1/3  "enable" %
%   B202:3/7  "trigger signal 6 leading edge os" %
%   L187:6  "ins 6 trigger count" %
% Rung: 20 %
SOR XIC B202:3/7 BST FFL N200:6 #N200:25 R6:1 4 0 NXB FFL 0 #L199:15 R6:2 4 0 BND EOR
%   B202:3/7  "trigger signal 6 leading edge os" %
%   N200:6  INS_6_TRIG_LOC %
%   N200:25  T6POS1 %
%   R6:1  "track part location untill acquire 6" %
%   L199:15  A6TM1 %
%   R6:2  "track acquire time 6" %

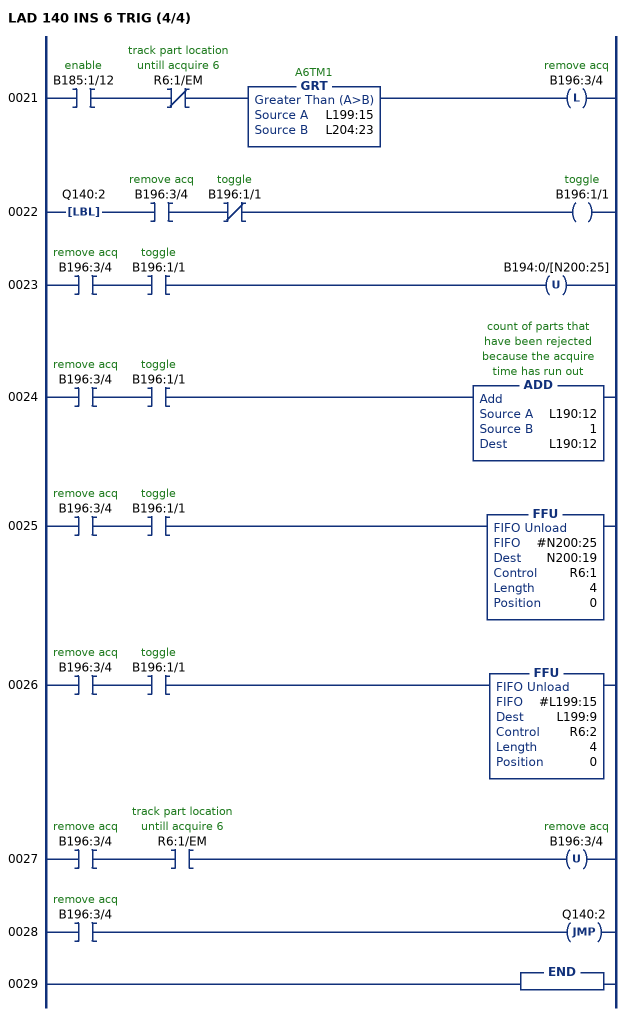
% Rung: 21 %
SOR XIC B185:1/12 XIO R6:1/EM GRT L199:15 L204:23 OTL B196:3/4 EOR
%   B185:1/12  "enable" %
%   R6:1  "track part location untill acquire 6" %
%   L199:15  A6TM1 %
%   B196:3/4  "remove acq" %
% Rung: 22 %
SOR LBL Q140:2 XIC B196:3/4 XIO B196:1/1 OTE B196:1/1 EOR
%   B196:3/4  "remove acq" %
%   B196:1/1  "toggle" %
% Rung: 23 %
SOR XIC B196:3/4 XIC B196:1/1 OTU B194:0/[N200:25] EOR
%   B196:3/4  "remove acq" %
%   B196:1/1  "toggle" %
%   N200:25  T6POS1 %
% Rung: 24 %
SOR XIC B196:3/4 XIC B196:1/1 ADD L190:12 1 L190:12 EOR
%   B196:3/4  "remove acq" %
%   B196:1/1  "toggle" %
%   L190:12  "count of parts that have been rejected because the acquire time has run out" %
% Rung: 25 %
SOR XIC B196:3/4 XIC B196:1/1 FFU #N200:25 N200:19 R6:1 4 0 EOR
%   B196:3/4  "remove acq" %
%   B196:1/1  "toggle" %
%   N200:25  T6POS1 %
%   R6:1  "track part location untill acquire 6" %
% Rung: 26 %
SOR XIC B196:3/4 XIC B196:1/1 FFU #L199:15 L199:9 R6:2 4 0 EOR
%   B196:3/4  "remove acq" %
%   B196:1/1  "toggle" %
%   L199:15  A6TM1 %
%   R6:2  "track acquire time 6" %
% Rung: 27 %
SOR XIC B196:3/4 XIC R6:1/EM OTU B196:3/4 EOR
%   B196:3/4  "remove acq" %
%   R6:1  "track part location untill acquire 6" %
% Rung: 28 %
SOR XIC B196:3/4 JMP Q140:2 EOR
%   B196:3/4  "remove acq" %
% Rung: 29 %
SOR END EOR

LADDER 141 "INS 6 RSLT"
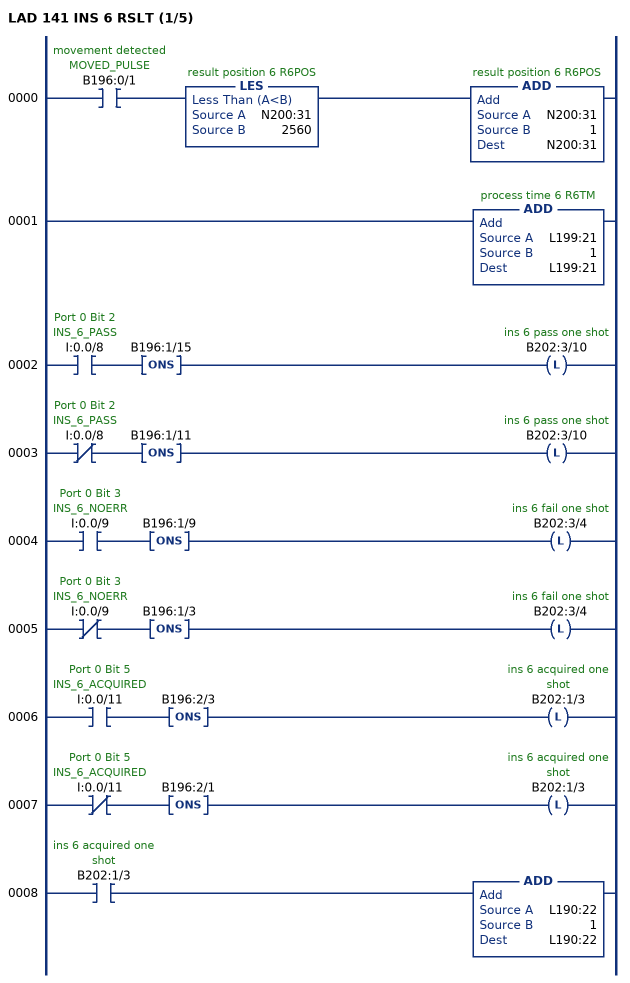
% Rung: 0 %
SOR XIC B196:0/1 LES N200:31 2560 ADD N200:31 1 N200:31 EOR
%   B196:0/1  MOVED_PULSE  "movement detected" %
%   N200:31  R6POS  "result position 6" %
% Rung: 1 %
SOR ADD L199:21 1 L199:21 EOR
%   L199:21  R6TM  "process time 6" %
% Rung: 2 %
SOR XIC I:0.0/8 ONS B196:1/15 OTL B202:3/10 EOR
%   I:0.0/8  INS_6_PASS  "Port 0 Bit 2" %
%   B202:3/10  "ins 6 pass one shot" %
% Rung: 3 %
SOR XIO I:0.0/8 ONS B196:1/11 OTL B202:3/10 EOR
%   I:0.0/8  INS_6_PASS  "Port 0 Bit 2" %
%   B202:3/10  "ins 6 pass one shot" %
% Rung: 4 %
SOR XIC I:0.0/9 ONS B196:1/9 OTL B202:3/4 EOR
%   I:0.0/9  INS_6_NOERR  "Port 0 Bit 3" %
%   B202:3/4  "ins 6 fail one shot" %
% Rung: 5 %
SOR XIO I:0.0/9 ONS B196:1/3 OTL B202:3/4 EOR
%   I:0.0/9  INS_6_NOERR  "Port 0 Bit 3" %
%   B202:3/4  "ins 6 fail one shot" %
% Rung: 6 %
SOR XIC I:0.0/11 ONS B196:2/3 OTL B202:1/3 EOR
%   I:0.0/11  INS_6_ACQUIRED  "Port 0 Bit 5" %
%   B202:1/3  "ins 6 acquired one shot" %
% Rung: 7 %
SOR XIO I:0.0/11 ONS B196:2/1 OTL B202:1/3 EOR
%   I:0.0/11  INS_6_ACQUIRED  "Port 0 Bit 5" %
%   B202:1/3  "ins 6 acquired one shot" %
% Rung: 8 %
SOR XIC B202:1/3 ADD L190:22 1 L190:22 EOR
%   B202:1/3  "ins 6 acquired one shot" %

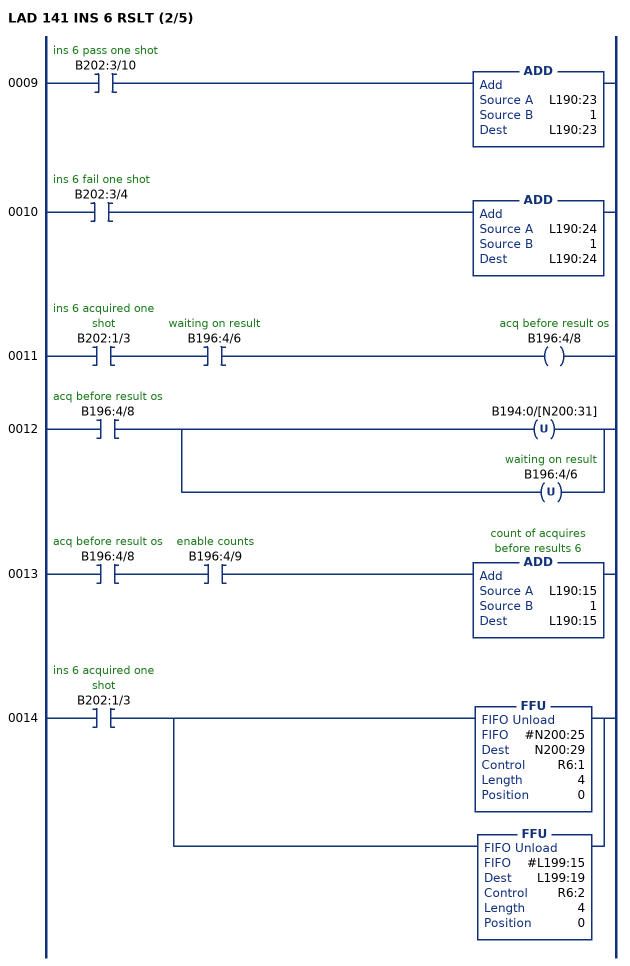
% Rung: 9 %
SOR XIC B202:3/10 ADD L190:23 1 L190:23 EOR
%   B202:3/10  "ins 6 pass one shot" %
% Rung: 10 %
SOR XIC B202:3/4 ADD L190:24 1 L190:24 EOR
%   B202:3/4  "ins 6 fail one shot" %
% Rung: 11 %
SOR XIC B202:1/3 XIC B196:4/6 OTE B196:4/8 EOR
%   B202:1/3  "ins 6 acquired one shot" %
%   B196:4/6  "waiting on result" %
%   B196:4/8  "acq before result os" %
% Rung: 12 %
SOR XIC B196:4/8 BST OTU B194:0/[N200:31] NXB OTU B196:4/6 BND EOR
%   B196:4/8  "acq before result os" %
%   N200:31  R6POS  "result position 6" %
%   B196:4/6  "waiting on result" %
% Rung: 13 %
SOR XIC B196:4/8 XIC B196:4/9 ADD L190:15 1 L190:15 EOR
%   B196:4/8  "acq before result os" %
%   B196:4/9  "enable counts" %
%   L190:15  "count of acquires before results 6" %
% Rung: 14 %
SOR XIC B202:1/3 BST FFU #N200:25 N200:29 R6:1 4 0 NXB FFU #L199:15 L199:19 R6:2 4 0 BND EOR
%   B202:1/3  "ins 6 acquired one shot" %
%   N200:25  T6POS1 %
%   R6:1  "track part location untill acquire 6" %
%   L199:15  A6TM1 %
%   R6:2  "track acquire time 6" %

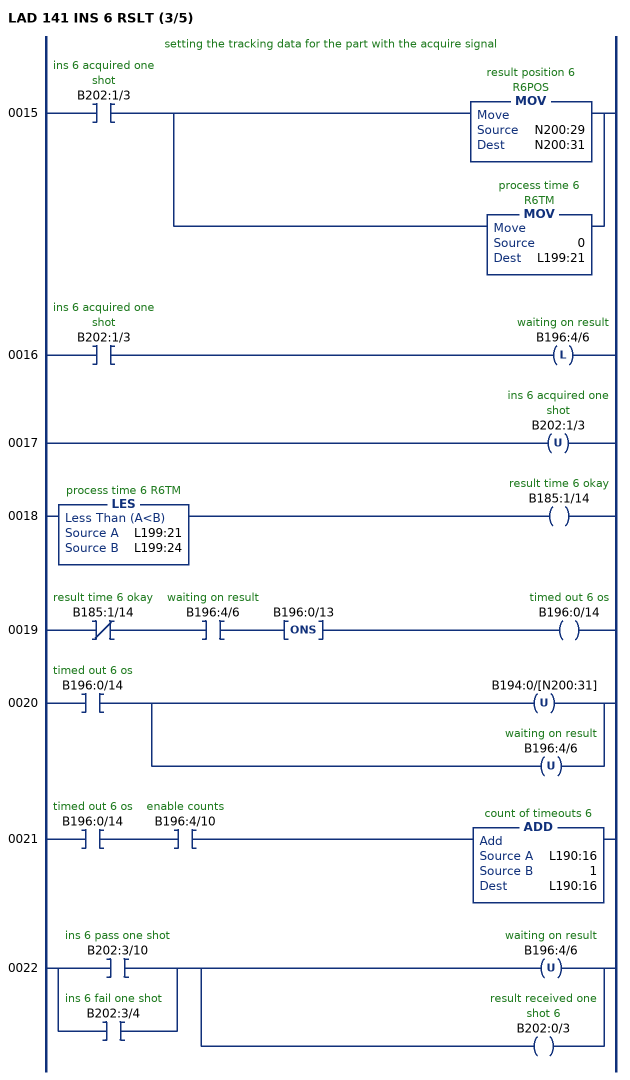
% Rung: 15 %
% setting the tracking data for the part with the acquire signal %
SOR XIC B202:1/3 BST MOV N200:29 N200:31 NXB MOV 0 L199:21 BND EOR
%   B202:1/3  "ins 6 acquired one shot" %
%   N200:31  R6POS  "result position 6" %
%   L199:21  R6TM  "process time 6" %
% Rung: 16 %
SOR XIC B202:1/3 OTL B196:4/6 EOR
%   B202:1/3  "ins 6 acquired one shot" %
%   B196:4/6  "waiting on result" %
% Rung: 17 %
SOR OTU B202:1/3 EOR
%   B202:1/3  "ins 6 acquired one shot" %
% Rung: 18 %
SOR LES L199:21 L199:24 OTE B185:1/14 EOR
%   L199:21  R6TM  "process time 6" %
%   B185:1/14  "result time 6 okay" %
% Rung: 19 %
SOR XIO B185:1/14 XIC B196:4/6 ONS B196:0/13 OTE B196:0/14 EOR
%   B185:1/14  "result time 6 okay" %
%   B196:4/6  "waiting on result" %
%   B196:0/14  "timed out 6 os" %
% Rung: 20 %
SOR XIC B196:0/14 BST OTU B194:0/[N200:31] NXB OTU B196:4/6 BND EOR
%   B196:0/14  "timed out 6 os" %
%   N200:31  R6POS  "result position 6" %
%   B196:4/6  "waiting on result" %
% Rung: 21 %
SOR XIC B196:0/14 XIC B196:4/10 ADD L190:16 1 L190:16 EOR
%   B196:0/14  "timed out 6 os" %
%   B196:4/10  "enable counts" %
%   L190:16  "count of timeouts 6" %
% Rung: 22 %
SOR BST XIC B202:3/10 NXB XIC B202:3/4 BND BST OTU B196:4/6 NXB OTE B202:0/3 BND EOR
%   B202:3/10  "ins 6 pass one shot" %
%   B202:3/4  "ins 6 fail one shot" %
%   B196:4/6  "waiting on result" %
%   B202:0/3  "result received one shot 6" %

